// TIA Portal V16 export
// export: Created 2024-06-24T15:42:28.6185009Z, ExportSetting WithDefaults, DisplayName Totally Integrated Automation Portal, DisplayVersion V16, DisplayName TIA Portal Version Control Interface, DisplayVersion V16, DisplayName TIA Portal Openness, DisplayVersion V16, DisplayName STEP 7 Professional, DisplayVersion V16, DisplayName STEP 7 Safety, DisplayVersion V16, DisplayName WinCC Advanced, DisplayVersion V16
DATA_BLOCK "DB_IO"   // DB1
{ S7_Optimized_Access := 'TRUE' }
VERSION : 0.1
// stored: AutoNumber true, IsOnlyStoredInLoadMemory false, IsRetainMemResEnabled false, IsWriteProtectedInAS false, MemoryReserve 100
   VAR
      One_shot : Array[0..10] of Bool;
      Green_position : DWord;
      Box_position : DWord;
      Green_raw_detected : Bool;
      System_running : Bool;
      StepA : Array[0..10] of Bool;
      Production_line_Init : Bool;
      System_Ready : Bool;
      Weight : Int;
      RunPickAndPlace : Bool;
      StepB : Array[0..10] of Bool;
      StepC : Array[0..10] of Bool;
      "counter" : Int;
   END_VAR
BEGIN
END_DATA_BLOCK
